Fanuc KAREL source: kt00554.KL

PROGRAM KT00554
%NOLOCKGROUP
VAR
V1 : VECTOR;V2 : VECTOR;OUT : VECTOR
BEGIN
--
--
V1.X=1.0
V2.Y=2.0
V1.X=1.0
V2.Y=2.0
OUT=(V1-V2)
END KT00554
